// TIA Portal V17 export
// export: Created 2023-02-14T02:49:31.9210298Z, ExportSetting WithDefaults, DisplayName Totally Integrated Automation Portal, DisplayVersion V17, DisplayName TIA Portal Openness, DisplayVersion V17, DisplayName TIA Portal Teamcenter Gateway, DisplayVersion V17, DisplayName TIA Portal Version Control Interface, DisplayVersion V17, DisplayName SINAMICS Startdrive Advanced, DisplayVersion V17, DisplayName SINAMICS Startdrive G130, G150, S120, S150, SINAMICS MV, S210, DisplayVersion V17, DisplayName SINAMICS Startdrive G110M, G120, G120C, G120D, G120P, G115D, DisplayVersion V17, DisplayName STEP 7 Professional, DisplayVersion V17, DisplayName STEP 7 Safety, DisplayVersion V17, DisplayName WinCC Professional, DisplayVersion V17
FUNCTION "IO MCC Preparation" : Void   // FC5, LAD
{ S7_Optimized_Access := 'TRUE' }
VERSION : 0.1
// stored: AutoNumber true, IsIECCheckEnabled false, SetENOAutomatically false, UDAEnableTagReadback false
BEGIN

REGION Network 1
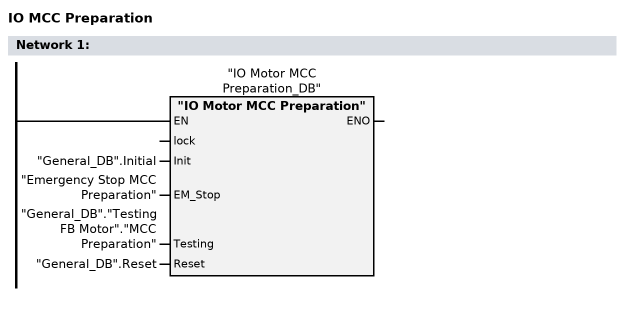
   RUNG wire#powerrail
      "IO Motor MCC Preparation_DB"(lock :=, Init := "General_DB".Initial, EM_Stop := "Emergency Stop MCC Preparation", Testing := "General_DB"."Testing FB Motor"."MCC Preparation", Reset := "General_DB".Reset)
   END_RUNG
   // the same network as SCL:
   "IO Motor MCC Preparation_DB"(Init := "General_DB".Initial,   // "IO Motor MCC Preparation"
                           EM_Stop := "Emergency Stop MCC Preparation",
                           Testing := "General_DB"."Testing FB Motor"."MCC Preparation",
                           Reset := "General_DB".Reset);
END_REGION
END_FUNCTION
